(* IEC 61131-3 sources: industrial-automation-plc-lab/analog-sensor-scaling/src, 2 files *)

(* ---- degs-function.st ---- *)
(* Declaration *)
FUNCTION degs : REAL
VAR_INPUT
	 temp_raw : UINT;

	rTmin : REAL;

	rTmax : REAL;
END_VAR
VAR
 iMin : INT ;

 iMax : INT ;
END_VAR

(* Implementation *)
iMin := 0;
iMax := 32767;
degs := rTmin + (UINT_TO_REAL(temp_raw) - INT_TO_REAL(iMin)) * (rTmax - rTmin) / (INT_TO_REAL(iMax) - INT_TO_REAL(iMin));

(* ---- plc-prg.st ---- *)
(* Declaration *)
PROGRAM PLC_PRG
VAR
    SensorTemp : UINT := 0;
    minSet : REAL := 20.0;
    maxSet : REAL := 100.0;
    measuredTemp : REAL;
END_VAR

(* Implementation *)
measuredTemp := degs(
    temp_raw := SensorTemp,
    rTmin := minSet,
    rTmax := maxSet
);
(* Execute Ladder Diagram program *)
PLC_PRG_LD();
